SYSTEM MechPress
  (* Version 1.0, Author, 4DIAC-Consortium *)
  APPLICATION Manual
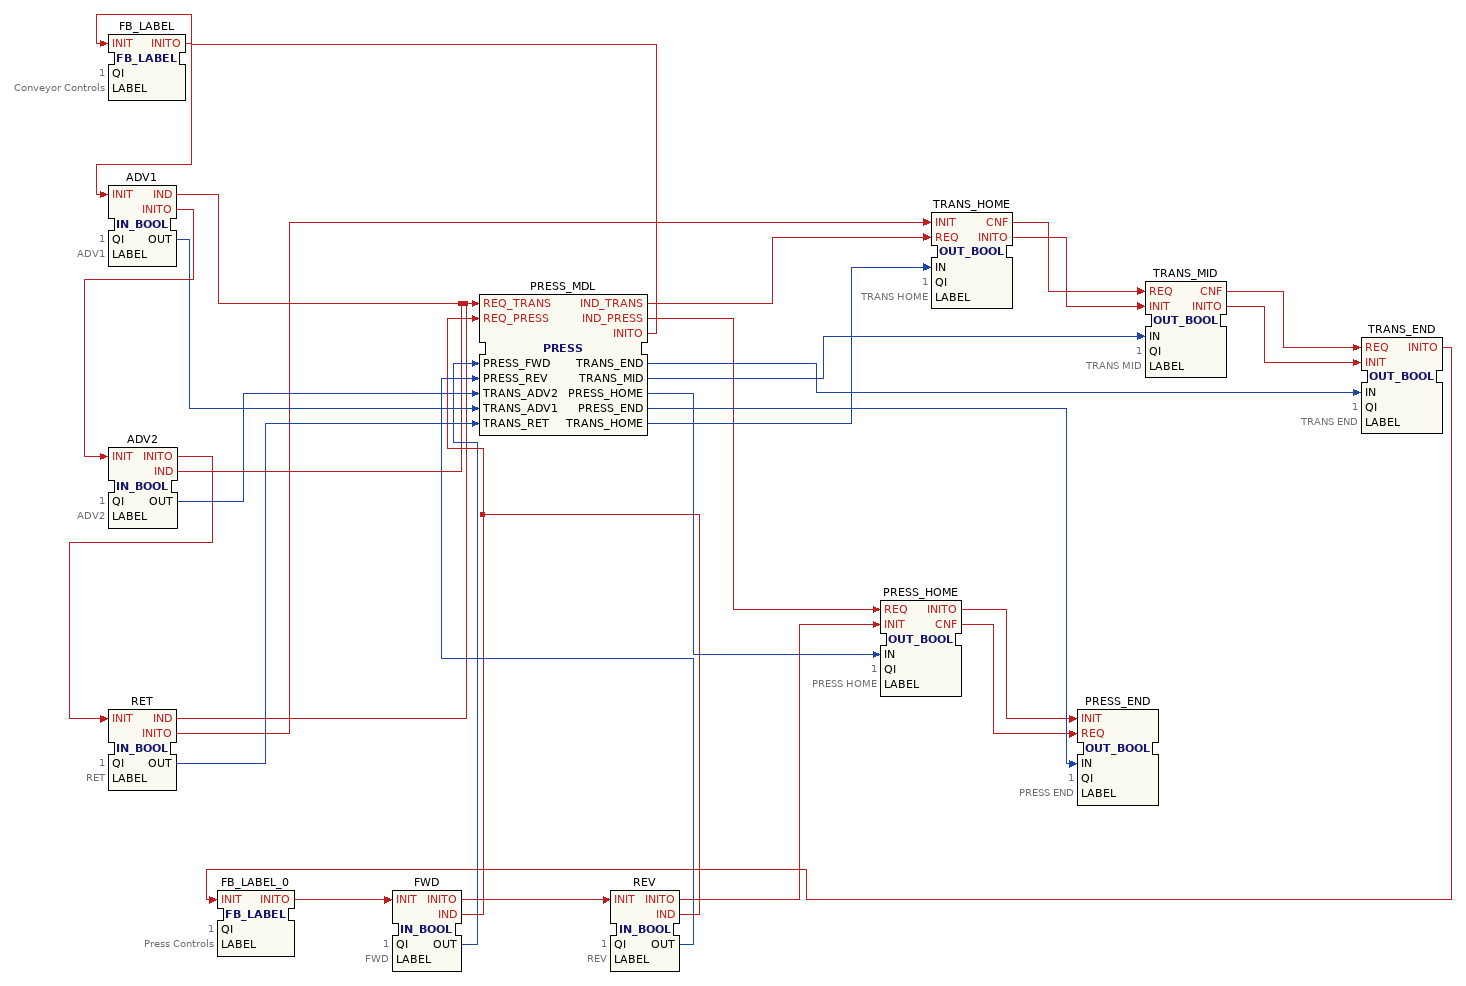
    FBS
      PRESS_MDL : PRESS;
      ADV1 : IN_BOOL(QI := 1, LABEL := ADV1);
      ADV2 : IN_BOOL(QI := 1, LABEL := ADV2);
      RET : IN_BOOL(QI := 1, LABEL := RET);
      FWD : IN_BOOL(QI := 1, LABEL := FWD);
      REV : IN_BOOL(QI := 1, LABEL := REV);
      TRANS_HOME : OUT_BOOL(QI := 1, LABEL := TRANS HOME);
      TRANS_MID : OUT_BOOL(QI := 1, LABEL := TRANS MID);
      TRANS_END : OUT_BOOL(QI := 1, LABEL := TRANS END);
      PRESS_HOME : OUT_BOOL(QI := 1, LABEL := PRESS HOME);
      PRESS_END : OUT_BOOL(QI := 1, LABEL := PRESS END);
      FB_LABEL : FB_LABEL(QI := 1, LABEL := Conveyor Controls);
      FB_LABEL_0 : FB_LABEL(QI := 1, LABEL := Press Controls);
    END_FBS
    EVENT_CONNECTIONS
      PRESS_HOME.INITO TO PRESS_END.INIT;
      ADV1.IND TO PRESS_MDL.REQ_TRANS;
      RET.IND TO PRESS_MDL.REQ_TRANS;
      TRANS_HOME.CNF TO TRANS_MID.REQ;
      ADV2.INITO TO RET.INIT;
      ADV2.IND TO PRESS_MDL.REQ_TRANS;
      TRANS_MID.CNF TO TRANS_END.REQ;
      ADV1.INITO TO ADV2.INIT;
      RET.INITO TO TRANS_HOME.INIT;
      TRANS_MID.INITO TO TRANS_END.INIT;
      TRANS_HOME.INITO TO TRANS_MID.INIT;
      FWD.INITO TO REV.INIT;
      PRESS_MDL.IND_TRANS TO TRANS_HOME.REQ;
      PRESS_MDL.IND_PRESS TO PRESS_HOME.REQ;
      FWD.IND TO PRESS_MDL.REQ_PRESS;
      REV.INITO TO PRESS_HOME.INIT;
      PRESS_HOME.CNF TO PRESS_END.REQ;
      REV.IND TO PRESS_MDL.REQ_PRESS;
      PRESS_MDL.INITO TO FB_LABEL.INIT;
      FB_LABEL.INITO TO ADV1.INIT;
      TRANS_END.INITO TO FB_LABEL_0.INIT;
      FB_LABEL_0.INITO TO FWD.INIT;
    END_CONNECTIONS
    DATA_CONNECTIONS
      PRESS_MDL.TRANS_END TO TRANS_END.IN;
      PRESS_MDL.TRANS_MID TO TRANS_MID.IN;
      PRESS_MDL.PRESS_HOME TO PRESS_HOME.IN;
      PRESS_MDL.PRESS_END TO PRESS_END.IN;
      FWD.OUT TO PRESS_MDL.PRESS_FWD;
      REV.OUT TO PRESS_MDL.PRESS_REV;
      ADV2.OUT TO PRESS_MDL.TRANS_ADV2;
      PRESS_MDL.TRANS_HOME TO TRANS_HOME.IN;
      ADV1.OUT TO PRESS_MDL.TRANS_ADV1;
      RET.OUT TO PRESS_MDL.TRANS_RET;
    END_CONNECTIONS
  END_APPLICATION
  APPLICATION Simulation
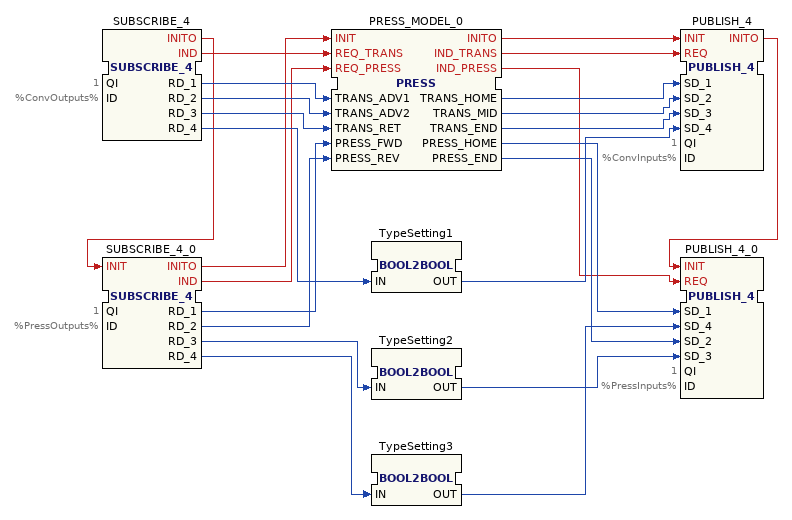
    FBS
      PRESS_MODEL_0 : PRESS;
      SUBSCRIBE_4 : SUBSCRIBE_4(QI := 1, ID := %ConvOutputs%);
      SUBSCRIBE_4_0 : SUBSCRIBE_4(QI := 1, ID := %PressOutputs%);
      TypeSetting1 : BOOL2BOOL;
      TypeSetting2 : BOOL2BOOL;
      TypeSetting3 : BOOL2BOOL;
      PUBLISH_4 : PUBLISH_4(QI := 1, ID := %ConvInputs%);
      PUBLISH_4_0 : PUBLISH_4(QI := 1, ID := %PressInputs%);
    END_FBS
    EVENT_CONNECTIONS
      SUBSCRIBE_4.INITO TO SUBSCRIBE_4_0.INIT;
      SUBSCRIBE_4_0.INITO TO PRESS_MODEL_0.INIT;
      SUBSCRIBE_4.IND TO PRESS_MODEL_0.REQ_TRANS;
      SUBSCRIBE_4_0.IND TO PRESS_MODEL_0.REQ_PRESS;
      PRESS_MODEL_0.INITO TO PUBLISH_4.INIT;
      PRESS_MODEL_0.IND_TRANS TO PUBLISH_4.REQ;
      PUBLISH_4.INITO TO PUBLISH_4_0.INIT;
      PRESS_MODEL_0.IND_PRESS TO PUBLISH_4_0.REQ;
    END_CONNECTIONS
    DATA_CONNECTIONS
      SUBSCRIBE_4.RD_1 TO PRESS_MODEL_0.TRANS_ADV1;
      SUBSCRIBE_4.RD_2 TO PRESS_MODEL_0.TRANS_ADV2;
      SUBSCRIBE_4.RD_3 TO PRESS_MODEL_0.TRANS_RET;
      SUBSCRIBE_4.RD_4 TO TypeSetting1.IN;
      SUBSCRIBE_4_0.RD_1 TO PRESS_MODEL_0.PRESS_FWD;
      SUBSCRIBE_4_0.RD_2 TO PRESS_MODEL_0.PRESS_REV;
      SUBSCRIBE_4_0.RD_3 TO TypeSetting2.IN;
      SUBSCRIBE_4_0.RD_4 TO TypeSetting3.IN;
      PRESS_MODEL_0.TRANS_HOME TO PUBLISH_4.SD_1;
      PRESS_MODEL_0.TRANS_MID TO PUBLISH_4.SD_2;
      PRESS_MODEL_0.TRANS_END TO PUBLISH_4.SD_3;
      TypeSetting1.OUT TO PUBLISH_4.SD_4;
      PRESS_MODEL_0.PRESS_HOME TO PUBLISH_4_0.SD_1;
      TypeSetting3.OUT TO PUBLISH_4_0.SD_4;
      PRESS_MODEL_0.PRESS_END TO PUBLISH_4_0.SD_2;
      TypeSetting2.OUT TO PUBLISH_4_0.SD_3;
    END_CONNECTIONS
  END_APPLICATION
  APPLICATION Automated
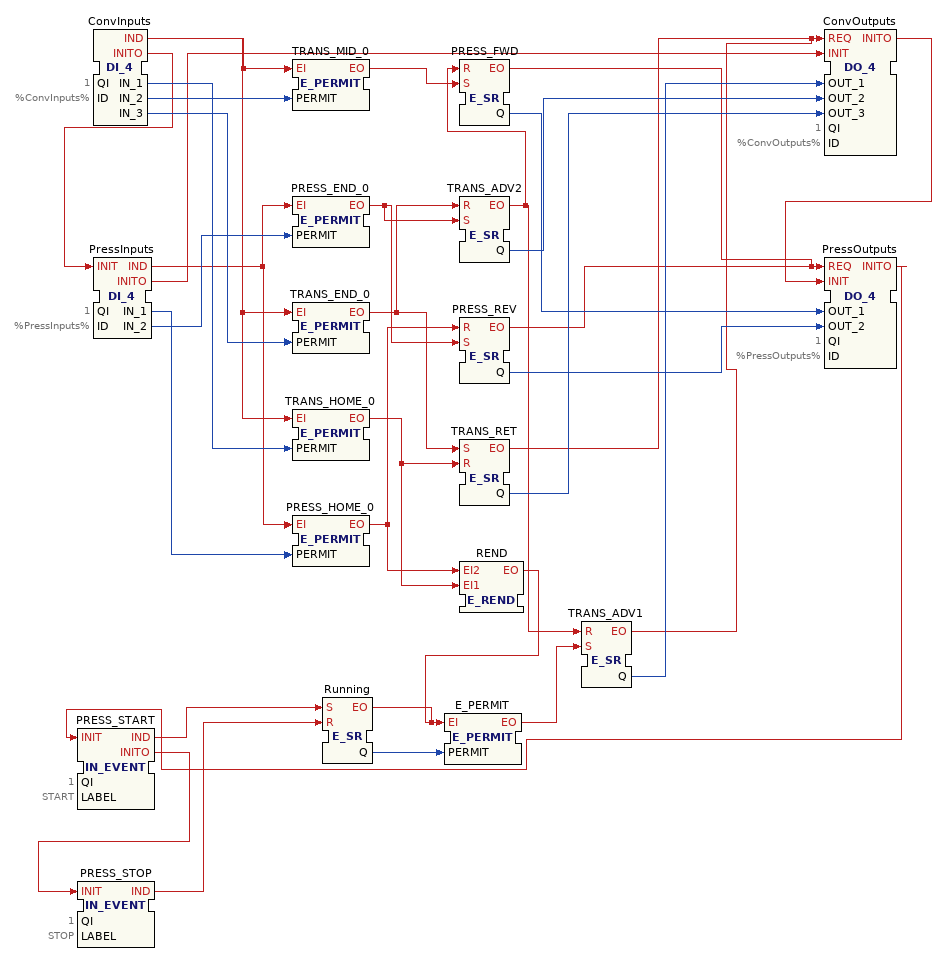
    FBS
      PRESS_START : IN_EVENT(QI := 1, LABEL := START);
      TRANS_MID_0 : E_PERMIT;
      PRESS_END_0 : E_PERMIT;
      TRANS_END_0 : E_PERMIT;
      TRANS_HOME_0 : E_PERMIT;
      PRESS_HOME_0 : E_PERMIT;
      PRESS_FWD : E_SR;
      TRANS_ADV2 : E_SR;
      PRESS_REV : E_SR;
      TRANS_RET : E_SR;
      TRANS_ADV1 : E_SR;
      REND : E_REND;
      ConvInputs : DI_4(QI := 1, ID := %ConvInputs%);
      PressInputs : DI_4(QI := 1, ID := %PressInputs%);
      ConvOutputs : DO_4(QI := 1, ID := %ConvOutputs%);
      PressOutputs : DO_4(QI := 1, ID := %PressOutputs%);
      Running : E_SR;
      E_PERMIT : E_PERMIT;
      PRESS_STOP : IN_EVENT(QI := 1, LABEL := STOP);
    END_FBS
    EVENT_CONNECTIONS
      PRESS_HOME_0.EO TO PRESS_REV.R;
      PRESS_HOME_0.EO TO REND.EI2;
      TRANS_ADV2.EO TO TRANS_ADV1.R;
      TRANS_HOME_0.EO TO REND.EI1;
      TRANS_ADV2.EO TO PRESS_FWD.R;
      TRANS_END_0.EO TO TRANS_ADV2.R;
      TRANS_MID_0.EO TO PRESS_FWD.S;
      TRANS_END_0.EO TO TRANS_RET.S;
      TRANS_HOME_0.EO TO TRANS_RET.R;
      PRESS_END_0.EO TO PRESS_REV.S;
      PRESS_END_0.EO TO TRANS_ADV2.S;
      ConvInputs.IND TO TRANS_MID_0.EI;
      ConvInputs.IND TO TRANS_END_0.EI;
      ConvInputs.IND TO TRANS_HOME_0.EI;
      PressInputs.IND TO PRESS_HOME_0.EI;
      PressInputs.IND TO PRESS_END_0.EI;
      TRANS_RET.EO TO ConvOutputs.REQ;
      TRANS_ADV1.EO TO ConvOutputs.REQ;
      PRESS_REV.EO TO PressOutputs.REQ;
      PRESS_FWD.EO TO PressOutputs.REQ;
      ConvInputs.INITO TO PressInputs.INIT;
      PressInputs.INITO TO ConvOutputs.INIT;
      ConvOutputs.INITO TO PressOutputs.INIT;
      PressOutputs.INITO TO PRESS_START.INIT;
      REND.EO TO E_PERMIT.EI;
      PRESS_START.IND TO Running.S;
      Running.EO TO E_PERMIT.EI;
      E_PERMIT.EO TO TRANS_ADV1.S;
      PRESS_START.INITO TO PRESS_STOP.INIT;
      PRESS_STOP.IND TO Running.R;
    END_CONNECTIONS
    DATA_CONNECTIONS
      ConvInputs.IN_1 TO TRANS_HOME_0.PERMIT;
      ConvInputs.IN_2 TO TRANS_MID_0.PERMIT;
      ConvInputs.IN_3 TO TRANS_END_0.PERMIT;
      PressInputs.IN_1 TO PRESS_HOME_0.PERMIT;
      PressInputs.IN_2 TO PRESS_END_0.PERMIT;
      TRANS_ADV1.Q TO ConvOutputs.OUT_1;
      TRANS_ADV2.Q TO ConvOutputs.OUT_2;
      TRANS_RET.Q TO ConvOutputs.OUT_3;
      PRESS_FWD.Q TO PressOutputs.OUT_1;
      PRESS_REV.Q TO PressOutputs.OUT_2;
      Running.Q TO E_PERMIT.PERMIT;
    END_CONNECTIONS
  END_APPLICATION
  APPLICATION Start
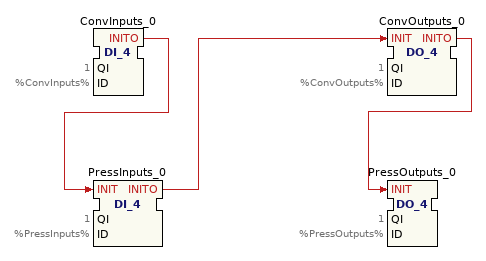
    FBS
      ConvInputs_0 : DI_4(QI := 1, ID := %ConvInputs%);
      PressInputs_0 : DI_4(QI := 1, ID := %PressInputs%);
      ConvOutputs_0 : DO_4(QI := 1, ID := %ConvOutputs%);
      PressOutputs_0 : DO_4(QI := 1, ID := %PressOutputs%);
    END_FBS
    EVENT_CONNECTIONS
      ConvOutputs_0.INITO TO PressOutputs_0.INIT;
      PressInputs_0.INITO TO ConvOutputs_0.INIT;
      ConvInputs_0.INITO TO PressInputs_0.INIT;
    END_CONNECTIONS
  END_APPLICATION
  DEVICE ManualTest : FBRT_WINDOW(BOUNDS := [100,100,360,280], GRID := [2,2], MGR_ID := "localhost:61500")
    {SET_ATTRIBUTE(Profile, HOLOBLOC)}
    RESOURCE Simulation : VIEW_PANEL(BKGD := COLOR#white, DIA := 25, SIZE := [7,4], VERTICAL := 0)
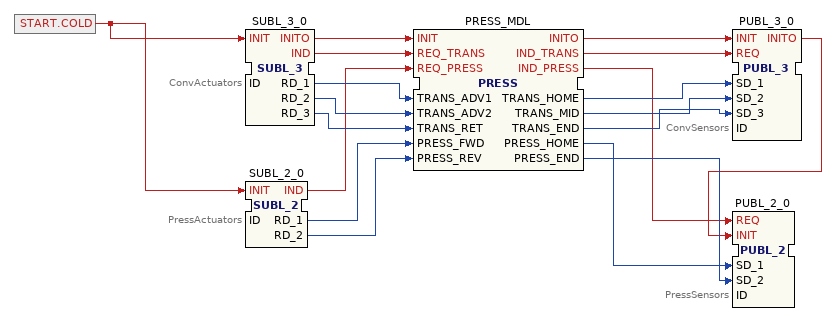
      FBS
        PRESS_MDL : PRESS;
        SUBL_3_0 : SUBL_3(ID := ConvActuators);
        PUBL_3_0 : PUBL_3(ID := ConvSensors);
        SUBL_2_0 : SUBL_2(ID := PressActuators);
        PUBL_2_0 : PUBL_2(ID := PressSensors);
      END_FBS
      EVENT_CONNECTIONS
        START.COLD TO SUBL_3_0.INIT;
        SUBL_3_0.INITO TO PRESS_MDL.INIT;
        SUBL_3_0.IND TO PRESS_MDL.REQ_TRANS;
        PRESS_MDL.INITO TO PUBL_3_0.INIT;
        PRESS_MDL.IND_TRANS TO PUBL_3_0.REQ;
        START.COLD TO SUBL_2_0.INIT;
        PRESS_MDL.IND_PRESS TO PUBL_2_0.REQ;
        PUBL_3_0.INITO TO PUBL_2_0.INIT;
        SUBL_2_0.IND TO PRESS_MDL.REQ_PRESS;
      END_CONNECTIONS
      DATA_CONNECTIONS
        SUBL_3_0.RD_1 TO PRESS_MDL.TRANS_ADV1;
        SUBL_3_0.RD_2 TO PRESS_MDL.TRANS_ADV2;
        SUBL_3_0.RD_3 TO PRESS_MDL.TRANS_RET;
        PRESS_MDL.TRANS_HOME TO PUBL_3_0.SD_1;
        PRESS_MDL.TRANS_MID TO PUBL_3_0.SD_2;
        PRESS_MDL.TRANS_END TO PUBL_3_0.SD_3;
        PRESS_MDL.PRESS_HOME TO PUBL_2_0.SD_1;
        PRESS_MDL.PRESS_END TO PUBL_2_0.SD_2;
        SUBL_2_0.RD_1 TO PRESS_MDL.PRESS_FWD;
        SUBL_2_0.RD_2 TO PRESS_MDL.PRESS_REV;
      END_CONNECTIONS
    END_RESOURCE
    RESOURCE PressControls : PANEL_RESOURCE(COLS := 1)
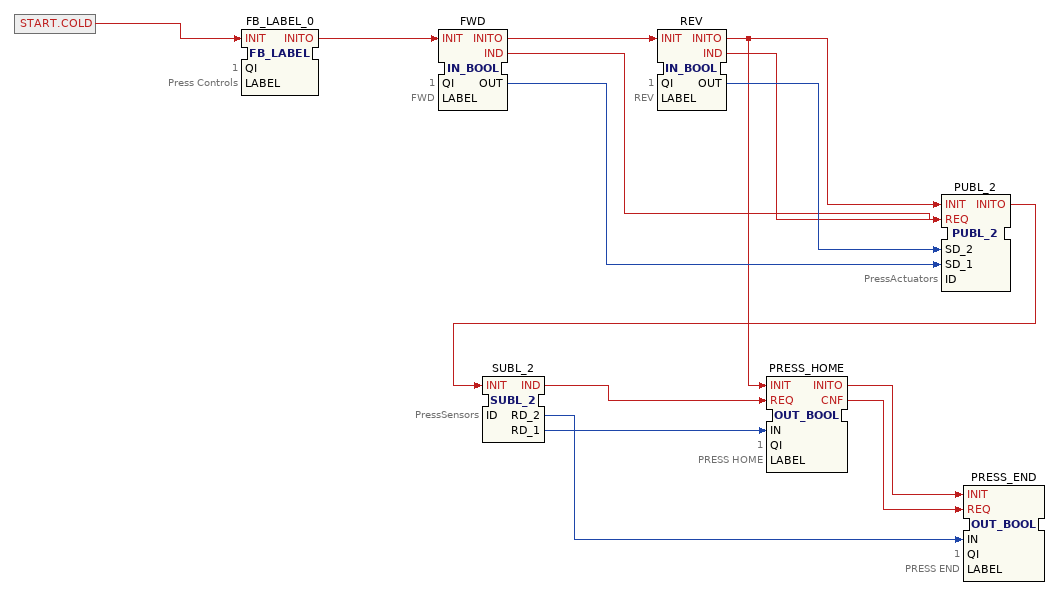
      FBS
        FWD : IN_BOOL(QI := 1, LABEL := FWD);
        REV : IN_BOOL(QI := 1, LABEL := REV);
        PRESS_HOME : OUT_BOOL(QI := 1, LABEL := PRESS HOME);
        PRESS_END : OUT_BOOL(QI := 1, LABEL := PRESS END);
        PUBL_2 : PUBL_2(ID := PressActuators);
        SUBL_2 : SUBL_2(ID := PressSensors);
        FB_LABEL_0 : FB_LABEL(QI := 1, LABEL := Press Controls);
      END_FBS
      EVENT_CONNECTIONS
        FWD.INITO TO REV.INIT;
        REV.INITO TO PRESS_HOME.INIT;
        PRESS_HOME.INITO TO PRESS_END.INIT;
        PRESS_HOME.CNF TO PRESS_END.REQ;
        REV.INITO TO PUBL_2.INIT;
        REV.IND TO PUBL_2.REQ;
        FWD.IND TO PUBL_2.REQ;
        SUBL_2.IND TO PRESS_HOME.REQ;
        PUBL_2.INITO TO SUBL_2.INIT;
        FB_LABEL_0.INITO TO FWD.INIT;
        START.COLD TO FB_LABEL_0.INIT;
      END_CONNECTIONS
      DATA_CONNECTIONS
        REV.OUT TO PUBL_2.SD_2;
        FWD.OUT TO PUBL_2.SD_1;
        SUBL_2.RD_2 TO PRESS_END.IN;
        SUBL_2.RD_1 TO PRESS_HOME.IN;
      END_CONNECTIONS
    END_RESOURCE
    RESOURCE ConveyorControls : PANEL_RESOURCE(COLS := 1)
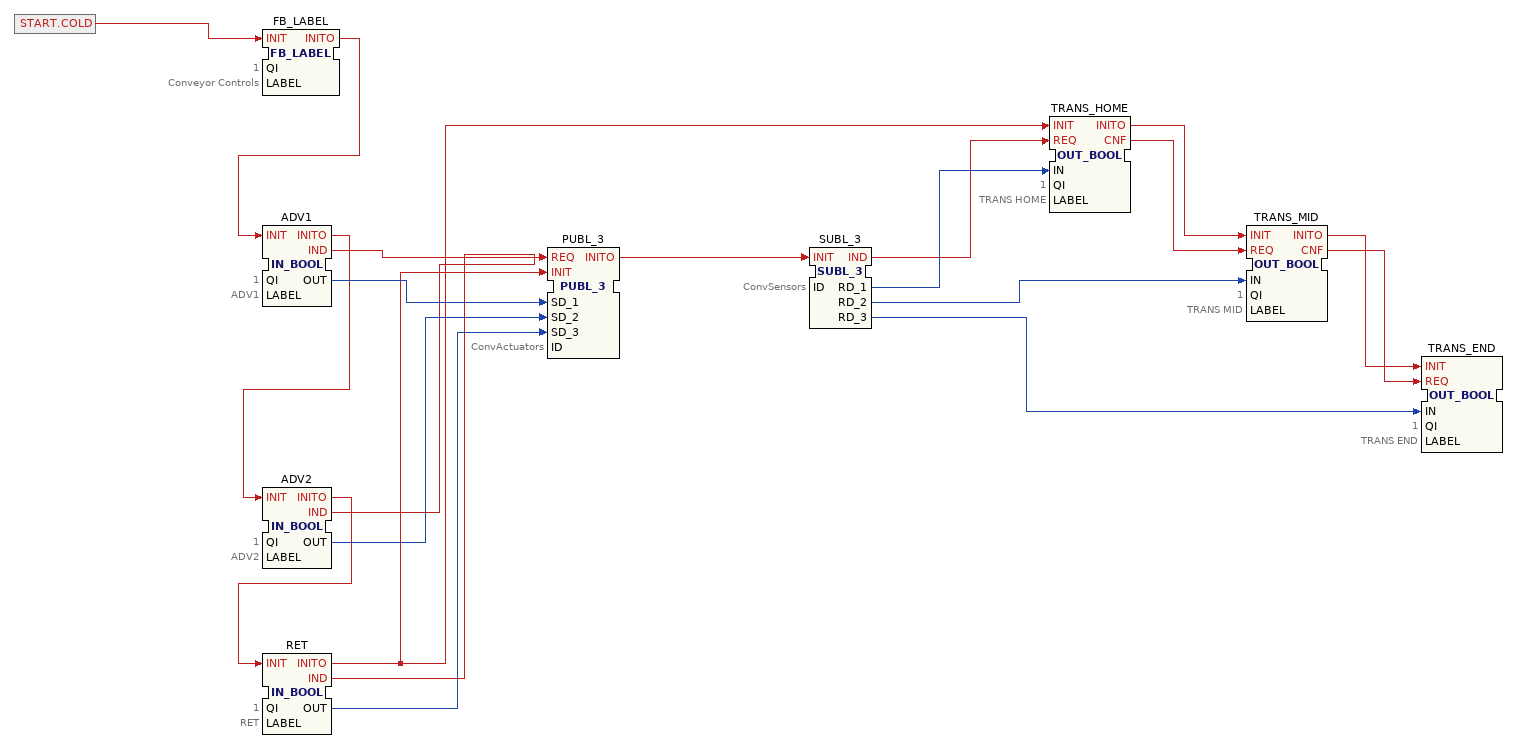
      FBS
        RET : IN_BOOL(QI := 1, LABEL := RET);
        ADV1 : IN_BOOL(QI := 1, LABEL := ADV1);
        ADV2 : IN_BOOL(QI := 1, LABEL := ADV2);
        TRANS_HOME : OUT_BOOL(QI := 1, LABEL := TRANS HOME);
        TRANS_MID : OUT_BOOL(QI := 1, LABEL := TRANS MID);
        TRANS_END : OUT_BOOL(QI := 1, LABEL := TRANS END);
        PUBL_3 : PUBL_3(ID := ConvActuators);
        SUBL_3 : SUBL_3(ID := ConvSensors);
        FB_LABEL : FB_LABEL(QI := 1, LABEL := Conveyor Controls);
      END_FBS
      EVENT_CONNECTIONS
        ADV1.INITO TO ADV2.INIT;
        ADV2.INITO TO RET.INIT;
        RET.INITO TO TRANS_HOME.INIT;
        TRANS_HOME.INITO TO TRANS_MID.INIT;
        TRANS_HOME.CNF TO TRANS_MID.REQ;
        TRANS_MID.INITO TO TRANS_END.INIT;
        TRANS_MID.CNF TO TRANS_END.REQ;
        ADV1.IND TO PUBL_3.REQ;
        ADV2.IND TO PUBL_3.REQ;
        RET.IND TO PUBL_3.REQ;
        RET.INITO TO PUBL_3.INIT;
        PUBL_3.INITO TO SUBL_3.INIT;
        SUBL_3.IND TO TRANS_HOME.REQ;
        FB_LABEL.INITO TO ADV1.INIT;
        START.COLD TO FB_LABEL.INIT;
      END_CONNECTIONS
      DATA_CONNECTIONS
        ADV1.OUT TO PUBL_3.SD_1;
        ADV2.OUT TO PUBL_3.SD_2;
        RET.OUT TO PUBL_3.SD_3;
        SUBL_3.RD_1 TO TRANS_HOME.IN;
        SUBL_3.RD_2 TO TRANS_MID.IN;
        SUBL_3.RD_3 TO TRANS_END.IN;
      END_CONNECTIONS
    END_RESOURCE
  END_DEVICE
  DEVICE Simulation : FBRT_WINDOW(BOUNDS := [0,0,177,158], MGR_ID := "localhost:61501")
    {SET_ATTRIBUTE(Profile, HOLOBLOC)}
    RESOURCE Simulation : VIEW_PANEL(DIA := 25, SIZE := [7,4], VERTICAL := 0)
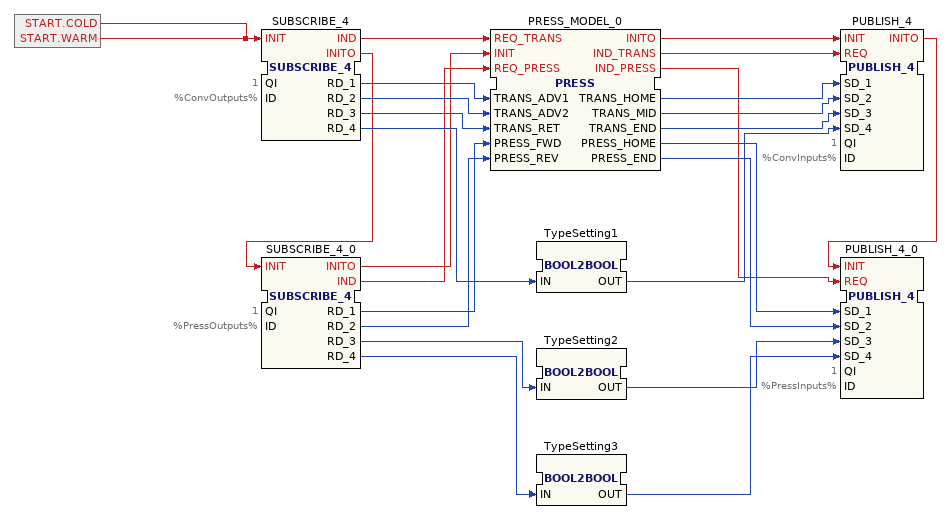
      FBS
        PRESS_MODEL_0 : PRESS;
        SUBSCRIBE_4 : SUBSCRIBE_4(QI := 1, ID := %ConvOutputs%);
        SUBSCRIBE_4_0 : SUBSCRIBE_4(QI := 1, ID := %PressOutputs%);
        TypeSetting1 : BOOL2BOOL;
        TypeSetting2 : BOOL2BOOL;
        TypeSetting3 : BOOL2BOOL;
        PUBLISH_4 : PUBLISH_4(QI := 1, ID := %ConvInputs%);
        PUBLISH_4_0 : PUBLISH_4(QI := 1, ID := %PressInputs%);
      END_FBS
      EVENT_CONNECTIONS
        SUBSCRIBE_4.IND TO PRESS_MODEL_0.REQ_TRANS;
        SUBSCRIBE_4.INITO TO SUBSCRIBE_4_0.INIT;
        SUBSCRIBE_4_0.INITO TO PRESS_MODEL_0.INIT;
        SUBSCRIBE_4_0.IND TO PRESS_MODEL_0.REQ_PRESS;
        PRESS_MODEL_0.INITO TO PUBLISH_4.INIT;
        PRESS_MODEL_0.IND_TRANS TO PUBLISH_4.REQ;
        PUBLISH_4.INITO TO PUBLISH_4_0.INIT;
        PRESS_MODEL_0.IND_PRESS TO PUBLISH_4_0.REQ;
        START.COLD TO SUBSCRIBE_4.INIT;
        START.WARM TO SUBSCRIBE_4.INIT;
      END_CONNECTIONS
      DATA_CONNECTIONS
        SUBSCRIBE_4.RD_1 TO PRESS_MODEL_0.TRANS_ADV1;
        SUBSCRIBE_4.RD_2 TO PRESS_MODEL_0.TRANS_ADV2;
        SUBSCRIBE_4.RD_3 TO PRESS_MODEL_0.TRANS_RET;
        SUBSCRIBE_4_0.RD_1 TO PRESS_MODEL_0.PRESS_FWD;
        SUBSCRIBE_4_0.RD_2 TO PRESS_MODEL_0.PRESS_REV;
        SUBSCRIBE_4.RD_4 TO TypeSetting1.IN;
        SUBSCRIBE_4_0.RD_3 TO TypeSetting2.IN;
        SUBSCRIBE_4_0.RD_4 TO TypeSetting3.IN;
        PRESS_MODEL_0.TRANS_HOME TO PUBLISH_4.SD_1;
        PRESS_MODEL_0.TRANS_MID TO PUBLISH_4.SD_2;
        PRESS_MODEL_0.TRANS_END TO PUBLISH_4.SD_3;
        TypeSetting1.OUT TO PUBLISH_4.SD_4;
        PRESS_MODEL_0.PRESS_HOME TO PUBLISH_4_0.SD_1;
        PRESS_MODEL_0.PRESS_END TO PUBLISH_4_0.SD_2;
        TypeSetting2.OUT TO PUBLISH_4_0.SD_3;
        TypeSetting3.OUT TO PUBLISH_4_0.SD_4;
      END_CONNECTIONS
    END_RESOURCE
  END_DEVICE
  DEVICE Control : FORTE_PC(MGR_ID := "localhost:61499")
    {SET_ATTRIBUTE(Profile, HOLOBLOC)}
    RESOURCE EMB_RES : EMB_RES
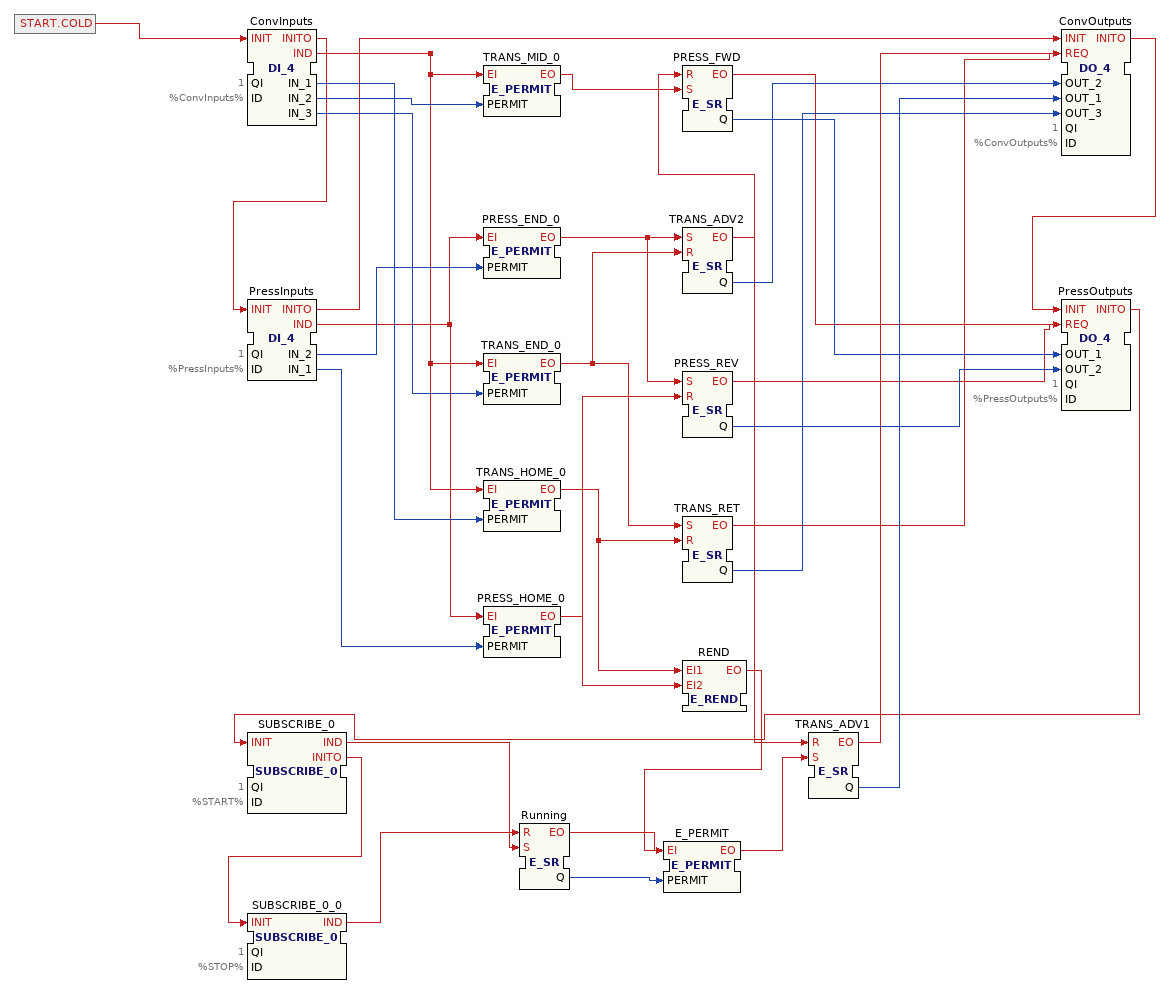
      FBS
        TRANS_HOME_0 : E_PERMIT;
        REND : E_REND;
        PressOutputs : DO_4(QI := 1, ID := %PressOutputs%);
        PressInputs : DI_4(QI := 1, ID := %PressInputs%);
        TRANS_ADV2 : E_SR;
        ConvOutputs : DO_4(QI := 1, ID := %ConvOutputs%);
        TRANS_ADV1 : E_SR;
        ConvInputs : DI_4(QI := 1, ID := %ConvInputs%);
        PRESS_FWD : E_SR;
        PRESS_END_0 : E_PERMIT;
        PRESS_REV : E_SR;
        TRANS_MID_0 : E_PERMIT;
        TRANS_END_0 : E_PERMIT;
        TRANS_RET : E_SR;
        PRESS_HOME_0 : E_PERMIT;
        Running : E_SR;
        E_PERMIT : E_PERMIT;
        SUBSCRIBE_0 : SUBSCRIBE_0(QI := 1, ID := %START%);
        SUBSCRIBE_0_0 : SUBSCRIBE_0(QI := 1, ID := %STOP%);
      END_FBS
      EVENT_CONNECTIONS
        TRANS_HOME_0.EO TO REND.EI1;
        PressInputs.INITO TO ConvOutputs.INIT;
        ConvOutputs.INITO TO PressOutputs.INIT;
        TRANS_ADV2.EO TO TRANS_ADV1.R;
        TRANS_ADV1.EO TO ConvOutputs.REQ;
        ConvInputs.INITO TO PressInputs.INIT;
        ConvInputs.IND TO TRANS_HOME_0.EI;
        TRANS_ADV2.EO TO PRESS_FWD.R;
        PRESS_FWD.EO TO PressOutputs.REQ;
        PressInputs.IND TO PRESS_END_0.EI;
        PRESS_END_0.EO TO TRANS_ADV2.S;
        PRESS_END_0.EO TO PRESS_REV.S;
        PRESS_REV.EO TO PressOutputs.REQ;
        ConvInputs.IND TO TRANS_MID_0.EI;
        TRANS_MID_0.EO TO PRESS_FWD.S;
        ConvInputs.IND TO TRANS_END_0.EI;
        TRANS_END_0.EO TO TRANS_ADV2.R;
        TRANS_END_0.EO TO TRANS_RET.S;
        TRANS_HOME_0.EO TO TRANS_RET.R;
        TRANS_RET.EO TO ConvOutputs.REQ;
        PressInputs.IND TO PRESS_HOME_0.EI;
        PRESS_HOME_0.EO TO PRESS_REV.R;
        PRESS_HOME_0.EO TO REND.EI2;
        START.COLD TO ConvInputs.INIT;
        REND.EO TO E_PERMIT.EI;
        Running.EO TO E_PERMIT.EI;
        E_PERMIT.EO TO TRANS_ADV1.S;
        PressOutputs.INITO TO SUBSCRIBE_0.INIT;
        SUBSCRIBE_0_0.IND TO Running.R;
        SUBSCRIBE_0.IND TO Running.S;
        SUBSCRIBE_0.INITO TO SUBSCRIBE_0_0.INIT;
      END_CONNECTIONS
      DATA_CONNECTIONS
        TRANS_ADV2.Q TO ConvOutputs.OUT_2;
        TRANS_ADV1.Q TO ConvOutputs.OUT_1;
        ConvInputs.IN_1 TO TRANS_HOME_0.PERMIT;
        PRESS_FWD.Q TO PressOutputs.OUT_1;
        PressInputs.IN_2 TO PRESS_END_0.PERMIT;
        PRESS_REV.Q TO PressOutputs.OUT_2;
        ConvInputs.IN_2 TO TRANS_MID_0.PERMIT;
        ConvInputs.IN_3 TO TRANS_END_0.PERMIT;
        TRANS_RET.Q TO ConvOutputs.OUT_3;
        PressInputs.IN_1 TO PRESS_HOME_0.PERMIT;
        Running.Q TO E_PERMIT.PERMIT;
      END_CONNECTIONS
    END_RESOURCE
  END_DEVICE
  DEVICE HMI : FBRT_WINDOW(BOUNDS := [300,0,55,108], MGR_ID := "localhost:61502")
    {SET_ATTRIBUTE(Profile, HOLOBLOC)}
    RESOURCE STARTSTOP : PANEL_RESOURCE(COLS := 1)
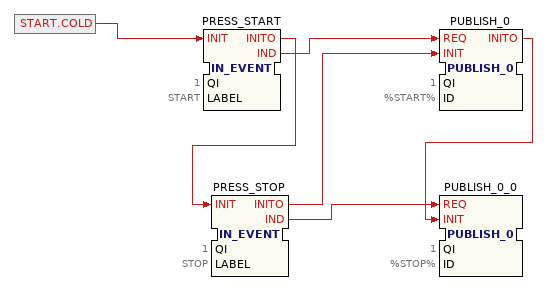
      FBS
        PRESS_START : IN_EVENT(QI := 1, LABEL := START);
        PRESS_STOP : IN_EVENT(QI := 1, LABEL := STOP);
        PUBLISH_0 : PUBLISH_0(QI := 1, ID := %START%);
        PUBLISH_0_0 : PUBLISH_0(QI := 1, ID := %STOP%);
      END_FBS
      EVENT_CONNECTIONS
        PRESS_START.INITO TO PRESS_STOP.INIT;
        START.COLD TO PRESS_START.INIT;
        PRESS_START.IND TO PUBLISH_0.REQ;
        PRESS_STOP.INITO TO PUBLISH_0.INIT;
        PRESS_STOP.IND TO PUBLISH_0_0.REQ;
        PUBLISH_0.INITO TO PUBLISH_0_0.INIT;
      END_CONNECTIONS
    END_RESOURCE
  END_DEVICE
  MAPPINGS
    Manual.PRESS_MDL ON ManualTest.Simulation.PRESS_MDL;
    Manual.ADV1 ON ManualTest.ConveyorControls.ADV1;
    Manual.ADV2 ON ManualTest.ConveyorControls.ADV2;
    Manual.RET ON ManualTest.ConveyorControls.RET;
    Manual.FWD ON ManualTest.PressControls.FWD;
    Manual.REV ON ManualTest.PressControls.REV;
    Manual.TRANS_HOME ON ManualTest.ConveyorControls.TRANS_HOME;
    Manual.TRANS_MID ON ManualTest.ConveyorControls.TRANS_MID;
    Manual.TRANS_END ON ManualTest.ConveyorControls.TRANS_END;
    Manual.PRESS_HOME ON ManualTest.PressControls.PRESS_HOME;
    Manual.PRESS_END ON ManualTest.PressControls.PRESS_END;
    Manual.FB_LABEL ON ManualTest.ConveyorControls.FB_LABEL;
    Manual.FB_LABEL_0 ON ManualTest.PressControls.FB_LABEL_0;
    Simulation.PRESS_MODEL_0 ON Simulation.Simulation.PRESS_MODEL_0;
    Simulation.SUBSCRIBE_4 ON Simulation.Simulation.SUBSCRIBE_4;
    Simulation.SUBSCRIBE_4_0 ON Simulation.Simulation.SUBSCRIBE_4_0;
    Simulation.TypeSetting1 ON Simulation.Simulation.TypeSetting1;
    Simulation.TypeSetting2 ON Simulation.Simulation.TypeSetting2;
    Simulation.TypeSetting3 ON Simulation.Simulation.TypeSetting3;
    Simulation.PUBLISH_4 ON Simulation.Simulation.PUBLISH_4;
    Simulation.PUBLISH_4_0 ON Simulation.Simulation.PUBLISH_4_0;
    Automated.PRESS_START ON HMI.STARTSTOP.PRESS_START;
    Automated.TRANS_MID_0 ON Control.EMB_RES.TRANS_MID_0;
    Automated.PRESS_END_0 ON Control.EMB_RES.PRESS_END_0;
    Automated.TRANS_END_0 ON Control.EMB_RES.TRANS_END_0;
    Automated.TRANS_HOME_0 ON Control.EMB_RES.TRANS_HOME_0;
    Automated.PRESS_HOME_0 ON Control.EMB_RES.PRESS_HOME_0;
    Automated.PRESS_FWD ON Control.EMB_RES.PRESS_FWD;
    Automated.TRANS_ADV2 ON Control.EMB_RES.TRANS_ADV2;
    Automated.PRESS_REV ON Control.EMB_RES.PRESS_REV;
    Automated.TRANS_RET ON Control.EMB_RES.TRANS_RET;
    Automated.TRANS_ADV1 ON Control.EMB_RES.TRANS_ADV1;
    Automated.REND ON Control.EMB_RES.REND;
    Automated.ConvInputs ON Control.EMB_RES.ConvInputs;
    Automated.PressInputs ON Control.EMB_RES.PressInputs;
    Automated.ConvOutputs ON Control.EMB_RES.ConvOutputs;
    Automated.PressOutputs ON Control.EMB_RES.PressOutputs;
    Automated.Running ON Control.EMB_RES.Running;
    Automated.E_PERMIT ON Control.EMB_RES.E_PERMIT;
    Automated.PRESS_STOP ON HMI.STARTSTOP.PRESS_STOP;
  END_MAPPINGS
  SEGMENTS
    Ethernet : Ethernet;
  END_SEGMENTS
  LINKS
    HMI => Ethernet;
    Control => Ethernet;
    Simulation => Ethernet;
  END_LINKS
END_SYSTEM
